// TIA Portal V21 export
FUNCTION_BLOCK "FB303"   // FB303, LAD
TITLE = FB303
{ S7_Optimized_Access := 'TRUE' }
AUTHOR : PRECISE
FAMILY : PRECISE
// SPARGING
// stored: AutoNumber false, MemoryReserve 100, SetENOAutomatically false
   VAR_INPUT
      Enable : Bool;
      Disable : Bool;
      Fault : Bool;
      SecPulse : Bool;
      AlwaysTrue { ExternalVisible := 'False'} : Bool;
      StartConfirmationPopupSel : Bool;   // StartConfirmationPopupSel: 0-NO/1-YES
      EndConfirmationPopupSel : Bool;   // EndConfirmationPopupSel: 0-NO/1-YES
      SpargingModeSel : Int;   // Sparging Mode Selection: 0-DO/1-Time
      SpargingTimebaseSel : Bool;   // Sparging Timebase Selection: 0-sec/1-min
      SpargingLineSel : Bool;   // Sparging LineSelection: 0-THRU GAS FILTER /1-THRU VV
      GasSel : Int;   // Gas Selection - 0-AIR/1-N2
      SetDO : Real := 10.0;   // For Sparging Mode Selection: 0-DO
      SpargingTimeMin : Int := 1;   // For Sparging Mode Selection: 1-Time & Sparging Timebase Selection: 1-min
      SpargingTimeSec : Int := 30;   // For Sparging Mode Selection: 1-Time & Sparging Timebase Selection: 0-sec
      PressuretoOpenVV : Real := 1.0;   // For Sparging LineSelection: 1-THRU VV
      PressuretoCloseVV : Real := 0.5;   // For Sparging LineSelection: 1-THRU VV
      ActualDO : Real;   // For Sparging Mode Selection: 0-DO
      ActualPressure : Real;   // For Sparging LineSelection: 1-THRU VV
      DelaytoOpenGasIn : Int := 3;
   END_VAR
   VAR_OUTPUT
      AirValve : Bool;
      N2Valve : Bool;
      SpargingLineValves : Bool;
      VentValve : Bool;   // For Sparging LineSelection: 1-THRU VV
      StartConfirmationPopup : Bool;   // For Start Confirmation Popup Selection: Yes
      EndConfirmationPopup : Bool;   // For End Confirmation Popup Selection: Yes
      SpargingTimeMinPV : DInt;
      SpargingTimeSecPV : DInt;
      PrintTrigger { ExternalAccessible := 'False'; ExternalVisible := 'False'; ExternalWritable := 'False'} : Bool;
      PrintWord : Int;
      PrintStatus : String[50];
   END_VAR
   VAR_IN_OUT
      Start : Bool;
      Stop : Bool;
      Reset : Bool;
      StartConfirmationAck : Bool;   // For Start Confirmation Popup Selection: Yes
      EndConfirmationAck : Bool;   // For End Confirmation Popup Selection: Yes
      SpareBtn1 : Bool;
      SpareBtn2 : Bool;
      SpareBtn3 : Bool;
      Running : Bool;
      Selected : Bool;
      Paused : Bool;
      StartConfirmationPopupTemp : Bool;   // For Start Confirmation Popup Selection: Yes
      EndConfirmationPopupTemp : Bool;   // For End Confirmation Popup Selection: Yes
      SpargingStarted : Bool;
      SpargingOver : Bool;
      SpargingTimerRunning : Bool;
   END_VAR
   VAR
      ValveOnDelayPV : Int;
      ValveOffDelayPV : Int;
      PrintTriggerTemp : Bool;
      RE1 : Bool;
      RE2 : Bool;
      RE3 : Bool;
      RE4 : Bool;
      RE5 : Bool;
      RE6 : Bool;
      RE7 : Bool;
      SpargingTimer : "FB101";
      PrintTriggerResetTimer { S7_SetPoint := 'True'} : TON_TIME;
      BtnResetTimer { S7_SetPoint := 'True'} : TON_TIME;
   END_VAR
   VAR_TEMP
      STATUS1 : String[40];
      STATUS2 : String[40];
      STATUS3 : String[40];
      STATUS4 : String[40];
      STATUS5 : String[40];
   END_VAR
   VAR_TEMP   // added for the SCL form of the ladder/FBD networks
      _w1 : Bool;
      _w2 : Bool;
      _w3 : Bool;
      _w4 : Bool;
      _w5 : Bool;
   END_VAR
BEGIN

REGION Network 1: Running
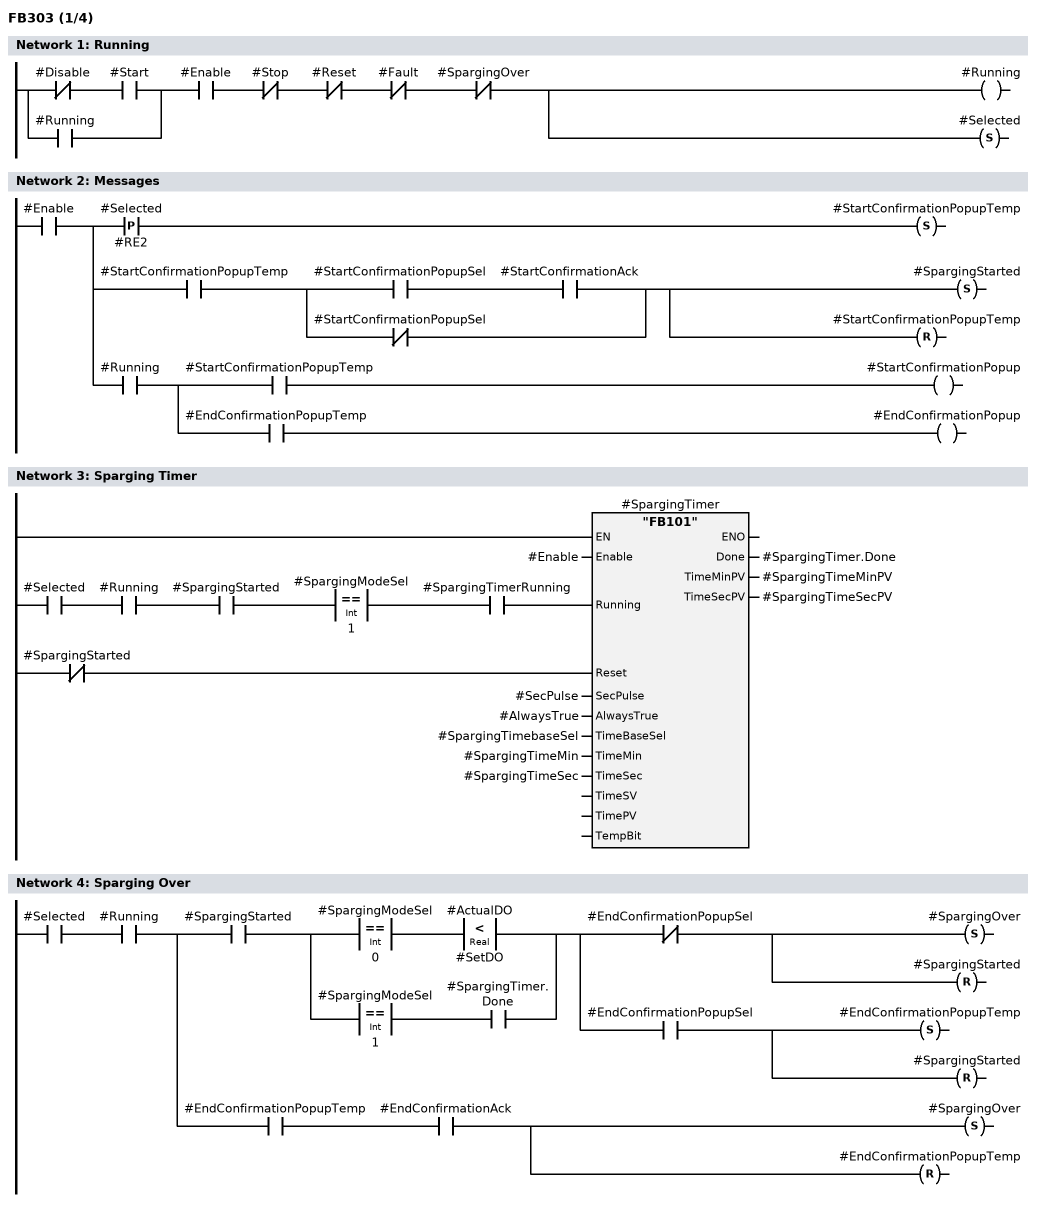
   RUNG wire#powerrail
      I_Contact( #Disable )
      Contact( #Start )
      wire#w1
      Contact( #Enable )
      I_Contact( #Stop )
      I_Contact( #Reset )
      I_Contact( #Fault )
      I_Contact( #SpargingOver )
      wire#w2
      Coil( #Running )
   END_RUNG
   RUNG wire#powerrail
      Contact( #Running )
   END_RUNG wire#w1
   RUNG wire#w2
      S_Coil( #Selected )
   END_RUNG
   // the same network as SCL:
   #Running := ((NOT #Disable AND #Start) OR #Running) AND #Enable AND NOT #Stop AND NOT #Reset AND NOT #Fault AND NOT #SpargingOver;
   IF #Running THEN #Selected := TRUE; END_IF;
END_REGION

REGION Network 2: Messages
   RUNG wire#powerrail
      Contact( #Enable )
      wire#w1
      P_Contact(operand := #Selected, bit := #RE2)
      S_Coil( #StartConfirmationPopupTemp )
   END_RUNG
   RUNG wire#w1
      Contact( #StartConfirmationPopupTemp )
      wire#w2
      Contact( #StartConfirmationPopupSel )
      Contact( #StartConfirmationAck )
      wire#w3
      S_Coil( #SpargingStarted )
   END_RUNG
   RUNG wire#w2
      I_Contact( #StartConfirmationPopupSel )
   END_RUNG wire#w3
   RUNG wire#w3
      R_Coil( #StartConfirmationPopupTemp )
   END_RUNG
   RUNG wire#w1
      Contact( #Running )
      wire#w4
      Contact( #StartConfirmationPopupTemp )
      Coil( #StartConfirmationPopup )
   END_RUNG
   RUNG wire#w4
      Contact( #EndConfirmationPopupTemp )
      Coil( #EndConfirmationPopup )
   END_RUNG
   // the same network as SCL:
   #_w1 := #Enable AND #Selected AND NOT #RE2;   // rising edge of #Selected
   #RE2 := #Selected;
   IF #_w1 THEN #StartConfirmationPopupTemp := TRUE; END_IF;
   IF #Enable AND #StartConfirmationPopupTemp AND ((#StartConfirmationPopupSel AND #StartConfirmationAck) OR NOT #StartConfirmationPopupSel) THEN
       #SpargingStarted := TRUE;
       #StartConfirmationPopupTemp := FALSE;
   END_IF;
   #_w2 := #Enable AND #Running;
   #StartConfirmationPopup := #_w2 AND #StartConfirmationPopupTemp;
   #EndConfirmationPopup := #_w2 AND #EndConfirmationPopupTemp;
END_REGION

REGION Network 3: Sparging Timer
   RUNG wire#powerrail
      #SpargingTimer(Running := wire#w1, Reset := wire#w2, Enable := #Enable, SecPulse := #SecPulse, AlwaysTrue := #AlwaysTrue, TimeBaseSel := #SpargingTimebaseSel, TimeMin := #SpargingTimeMin, TimeSec := #SpargingTimeSec, TimeSV :=, TimePV :=, TempBit :=, Done => #SpargingTimer.Done, TimeMinPV => #SpargingTimeMinPV, TimeSecPV => #SpargingTimeSecPV)
   END_RUNG
   RUNG wire#powerrail
      Contact( #Selected )
      Contact( #Running )
      Contact( #SpargingStarted )
      { S7_Templates := "SrcType := Int" } EQ_Contact(in1 := #SpargingModeSel, in2 := 1)
      Contact( #SpargingTimerRunning )
   END_RUNG wire#w1
   RUNG wire#powerrail
      I_Contact( #SpargingStarted )
   END_RUNG wire#w2
   // the same network as SCL:
   #SpargingTimer(Enable := #Enable,   // "FB101"
                  Running := #Selected AND #Running AND #SpargingStarted AND (#SpargingModeSel = 1) AND #SpargingTimerRunning,
                  Reset := NOT #SpargingStarted,
                  SecPulse := #SecPulse,
                  AlwaysTrue := #AlwaysTrue,
                  TimeBaseSel := #SpargingTimebaseSel,
                  TimeMin := #SpargingTimeMin,
                  TimeSec := #SpargingTimeSec,
                  Done => #SpargingTimer.Done,
                  TimeMinPV => #SpargingTimeMinPV,
                  TimeSecPV => #SpargingTimeSecPV);
END_REGION

REGION Network 4: Sparging Over
   RUNG wire#powerrail
      Contact( #Selected )
      Contact( #Running )
      wire#w1
      Contact( #SpargingStarted )
      wire#w2
      { S7_Templates := "SrcType := Int" } EQ_Contact(in1 := #SpargingModeSel, in2 := 0)
      { S7_Templates := "SrcType := Real" } LT_Contact(in1 := #ActualDO, in2 := #SetDO)
      wire#w3
      I_Contact( #EndConfirmationPopupSel )
      wire#w4
      S_Coil( #SpargingOver )
   END_RUNG
   RUNG wire#w2
      { S7_Templates := "SrcType := Int" } EQ_Contact(in1 := #SpargingModeSel, in2 := 1)
      Contact( #SpargingTimer.Done )
   END_RUNG wire#w3
   RUNG wire#w4
      R_Coil( #SpargingStarted )
   END_RUNG
   RUNG wire#w3
      Contact( #EndConfirmationPopupSel )
      wire#w5
      S_Coil( #EndConfirmationPopupTemp )
   END_RUNG
   RUNG wire#w5
      R_Coil( #SpargingStarted )
   END_RUNG
   RUNG wire#w1
      Contact( #EndConfirmationPopupTemp )
      Contact( #EndConfirmationAck )
      wire#w6
      S_Coil( #SpargingOver )
   END_RUNG
   RUNG wire#w6
      R_Coil( #EndConfirmationPopupTemp )
   END_RUNG
   // the same network as SCL:
   #_w1 := #Selected AND #Running;
   #_w2 := #_w1 AND #SpargingStarted AND (((#SpargingModeSel = 0) AND (#ActualDO < #SetDO)) OR ((#SpargingModeSel = 1) AND #SpargingTimer.Done));
   IF #_w2 AND NOT #EndConfirmationPopupSel THEN
       #SpargingOver := TRUE;
       #SpargingStarted := FALSE;
   END_IF;
   IF #_w2 AND #EndConfirmationPopupSel THEN
       #EndConfirmationPopupTemp := TRUE;
       #SpargingStarted := FALSE;
   END_IF;
   IF #_w1 AND #EndConfirmationPopupTemp AND #EndConfirmationAck THEN
       #SpargingOver := TRUE;
       #EndConfirmationPopupTemp := FALSE;
   END_IF;
END_REGION

REGION Network 5: Output On
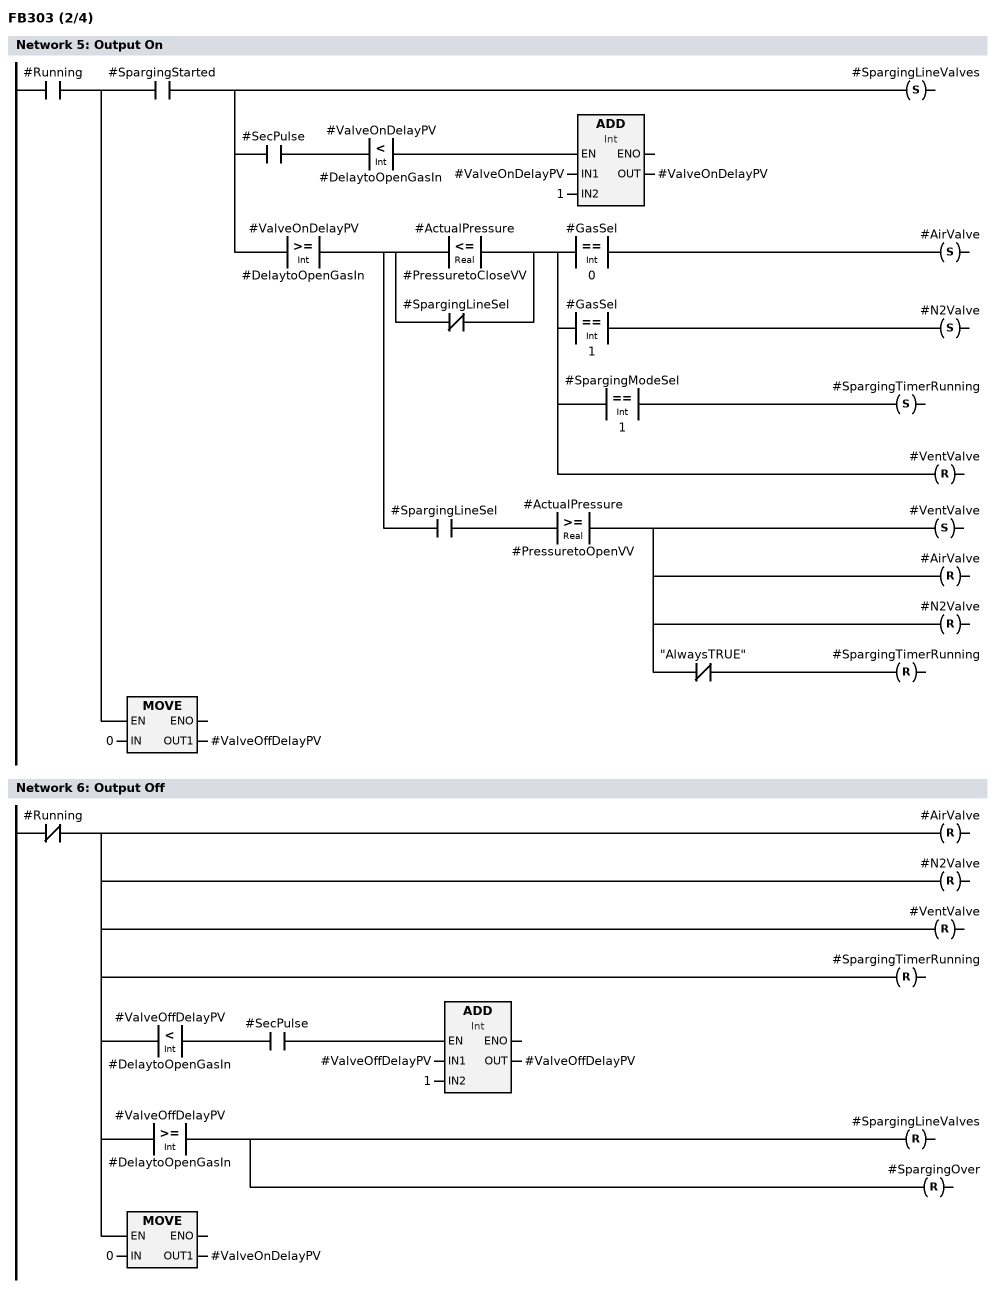
   RUNG wire#powerrail
      Contact( #Running )
      wire#w1
      Contact( #SpargingStarted )
      wire#w2
      S_Coil( #SpargingLineValves )
   END_RUNG
   RUNG wire#w2
      Contact( #SecPulse )
      { S7_Templates := "SrcType := Int" } LT_Contact(in1 := #ValveOnDelayPV, in2 := #DelaytoOpenGasIn)
      { S7_Templates := "SrcType := Int"; S7_GenerateENO := "TRUE" } Add(in1 := #ValveOnDelayPV, in2 := 1, out => #ValveOnDelayPV)
   END_RUNG
   RUNG wire#w2
      { S7_Templates := "SrcType := Int" } GE_Contact(in1 := #ValveOnDelayPV, in2 := #DelaytoOpenGasIn)
      wire#w3
      { S7_Templates := "SrcType := Real" } LE_Contact(in1 := #ActualPressure, in2 := #PressuretoCloseVV)
      wire#w4
      { S7_Templates := "SrcType := Int" } EQ_Contact(in1 := #GasSel, in2 := 0)
      S_Coil( #AirValve )
   END_RUNG
   RUNG wire#w3
      I_Contact( #SpargingLineSel )
   END_RUNG wire#w4
   RUNG wire#w4
      { S7_Templates := "SrcType := Int" } EQ_Contact(in1 := #GasSel, in2 := 1)
      S_Coil( #N2Valve )
   END_RUNG
   RUNG wire#w4
      { S7_Templates := "SrcType := Int" } EQ_Contact(in1 := #SpargingModeSel, in2 := 1)
      S_Coil( #SpargingTimerRunning )
   END_RUNG
   RUNG wire#w4
      R_Coil( #VentValve )
   END_RUNG
   RUNG wire#w3
      Contact( #SpargingLineSel )
      { S7_Templates := "SrcType := Real" } GE_Contact(in1 := #ActualPressure, in2 := #PressuretoOpenVV)
      wire#w5
      S_Coil( #VentValve )
   END_RUNG
   RUNG wire#w5
      R_Coil( #AirValve )
   END_RUNG
   RUNG wire#w5
      R_Coil( #N2Valve )
   END_RUNG
   RUNG wire#w5
      I_Contact( "AlwaysTRUE" )
      R_Coil( #SpargingTimerRunning )
   END_RUNG
   RUNG wire#w1
      { S7_GenerateENO := "TRUE" } Move(in := 0, out1 => #ValveOffDelayPV)
   END_RUNG
   // the same network as SCL:
   #_w1 := #Running AND #SpargingStarted;
   IF #_w1 THEN #SpargingLineValves := TRUE; END_IF;
   IF #_w1 AND #SecPulse AND (#ValveOnDelayPV < #DelaytoOpenGasIn) THEN
       #ValveOnDelayPV := #ValveOnDelayPV + 1;
   END_IF;
   #_w2 := #_w1 AND (#ValveOnDelayPV >= #DelaytoOpenGasIn);
   #_w3 := #_w2 AND ((#ActualPressure <= #PressuretoCloseVV) OR NOT #SpargingLineSel);
   IF #_w3 AND (#GasSel = 0) THEN #AirValve := TRUE; END_IF;
   IF #_w3 AND (#GasSel = 1) THEN #N2Valve := TRUE; END_IF;
   IF #_w3 AND (#SpargingModeSel = 1) THEN #SpargingTimerRunning := TRUE; END_IF;
   IF #_w3 THEN #VentValve := FALSE; END_IF;
   #_w4 := #_w2 AND #SpargingLineSel AND (#ActualPressure >= #PressuretoOpenVV);
   IF #_w4 THEN
       #VentValve := TRUE;
       #AirValve := FALSE;
       #N2Valve := FALSE;
   END_IF;
   IF #_w4 AND NOT "AlwaysTRUE" THEN #SpargingTimerRunning := FALSE; END_IF;
   IF #Running THEN #ValveOffDelayPV := 0; END_IF;
END_REGION

REGION Network 6: Output Off
   RUNG wire#powerrail
      I_Contact( #Running )
      wire#w1
      R_Coil( #AirValve )
   END_RUNG
   RUNG wire#w1
      R_Coil( #N2Valve )
   END_RUNG
   RUNG wire#w1
      R_Coil( #VentValve )
   END_RUNG
   RUNG wire#w1
      R_Coil( #SpargingTimerRunning )
   END_RUNG
   RUNG wire#w1
      { S7_Templates := "SrcType := Int" } LT_Contact(in1 := #ValveOffDelayPV, in2 := #DelaytoOpenGasIn)
      Contact( #SecPulse )
      { S7_Templates := "SrcType := Int"; S7_GenerateENO := "TRUE" } Add(in1 := #ValveOffDelayPV, in2 := 1, out => #ValveOffDelayPV)
   END_RUNG
   RUNG wire#w1
      { S7_Templates := "SrcType := Int" } GE_Contact(in1 := #ValveOffDelayPV, in2 := #DelaytoOpenGasIn)
      wire#w2
      R_Coil( #SpargingLineValves )
   END_RUNG
   RUNG wire#w2
      R_Coil( #SpargingOver )
   END_RUNG
   RUNG wire#w1
      { S7_GenerateENO := "TRUE" } Move(in := 0, out1 => #ValveOnDelayPV)
   END_RUNG
   // the same network as SCL:
   IF NOT #Running THEN
       #AirValve := FALSE;
       #N2Valve := FALSE;
       #VentValve := FALSE;
       #SpargingTimerRunning := FALSE;
   END_IF;
   IF NOT #Running AND (#ValveOffDelayPV < #DelaytoOpenGasIn) AND #SecPulse THEN
       #ValveOffDelayPV := #ValveOffDelayPV + 1;
   END_IF;
   IF NOT #Running AND (#ValveOffDelayPV >= #DelaytoOpenGasIn) THEN
       #SpargingLineValves := FALSE;
       #SpargingOver := FALSE;
   END_IF;
   IF NOT #Running THEN #ValveOnDelayPV := 0; END_IF;
END_REGION

REGION Network 7: Event Status
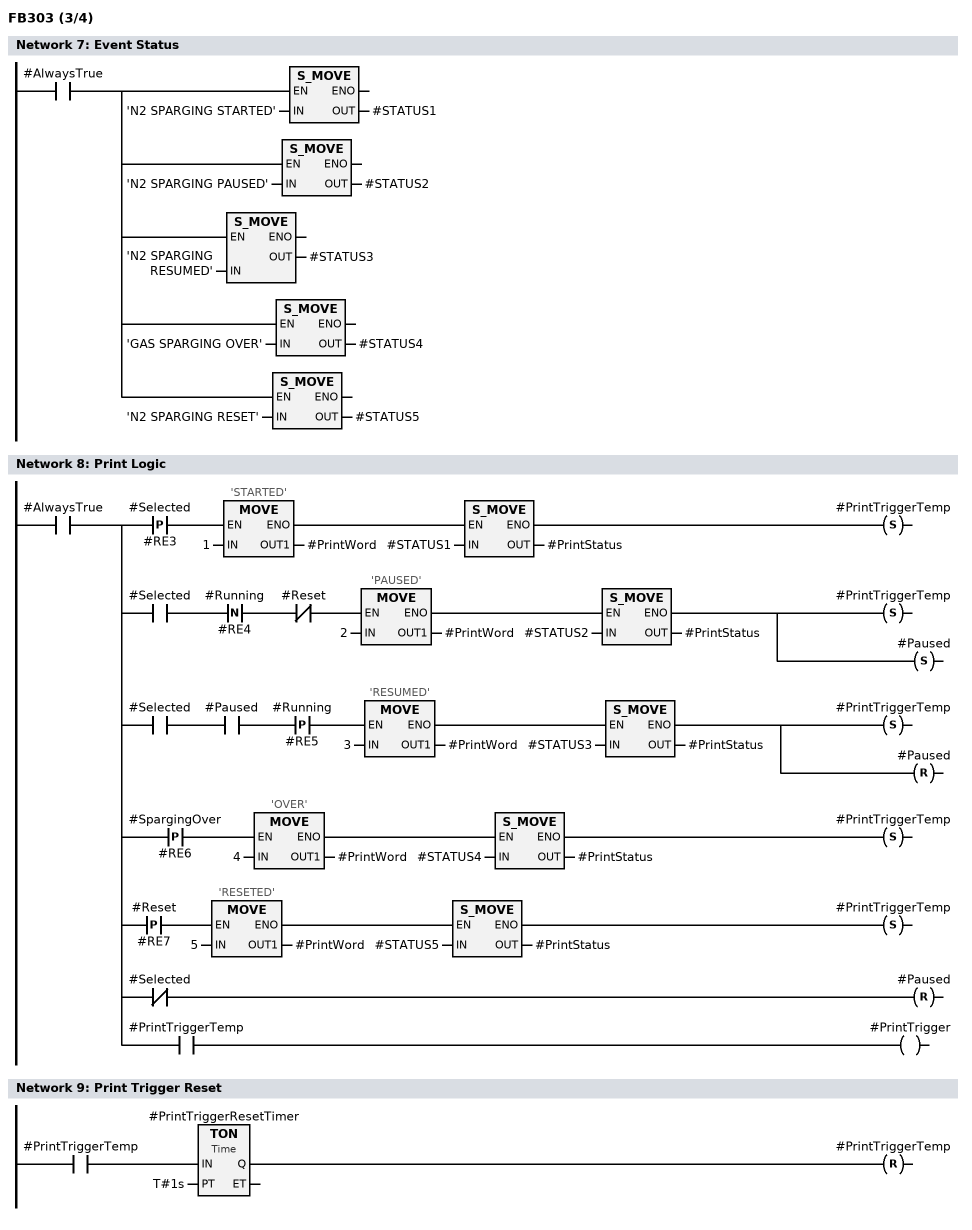
   RUNG wire#powerrail
      Contact( #AlwaysTrue )
      wire#w1
      S_Move(in := 'N2 SPARGING STARTED', out => #STATUS1)
   END_RUNG
   RUNG wire#w1
      S_Move(in := 'N2 SPARGING PAUSED', out => #STATUS2)
   END_RUNG
   RUNG wire#w1
      S_Move(in := 'N2 SPARGING RESUMED', out => #STATUS3)
   END_RUNG
   RUNG wire#w1
      S_Move(in := 'GAS SPARGING OVER', out => #STATUS4)
   END_RUNG
   RUNG wire#w1
      S_Move(in := 'N2 SPARGING RESET', out => #STATUS5)
   END_RUNG
   // the same network as SCL:
   IF #AlwaysTrue THEN
       #STATUS1 := 'N2 SPARGING STARTED';
       #STATUS2 := 'N2 SPARGING PAUSED';
       #STATUS3 := 'N2 SPARGING RESUMED';
       #STATUS4 := 'GAS SPARGING OVER';
       #STATUS5 := 'N2 SPARGING RESET';
   END_IF;
END_REGION

REGION Network 8: Print Logic
   RUNG wire#powerrail
      Contact( #AlwaysTrue )
      wire#w1
      P_Contact(operand := #Selected, bit := #RE3)
      { S7_GenerateENO := "TRUE" } Move(in := 1, out1 => #PrintWord)   // 'STARTED'
      S_Move(in := #STATUS1, out => #PrintStatus)
      S_Coil( #PrintTriggerTemp )
   END_RUNG
   RUNG wire#w1
      Contact( #Selected )
      N_Contact(operand := #Running, bit := #RE4)
      I_Contact( #Reset )
      { S7_GenerateENO := "TRUE" } Move(in := 2, out1 => #PrintWord)   // 'PAUSED'
      S_Move(in := #STATUS2, out => #PrintStatus)
      wire#w2
      S_Coil( #PrintTriggerTemp )
   END_RUNG
   RUNG wire#w2
      S_Coil( #Paused )
   END_RUNG
   RUNG wire#w1
      Contact( #Selected )
      Contact( #Paused )
      P_Contact(operand := #Running, bit := #RE5)
      { S7_GenerateENO := "TRUE" } Move(in := 3, out1 => #PrintWord)   // 'RESUMED'
      S_Move(in := #STATUS3, out => #PrintStatus)
      wire#w3
      S_Coil( #PrintTriggerTemp )
   END_RUNG
   RUNG wire#w3
      R_Coil( #Paused )
   END_RUNG
   RUNG wire#w1
      P_Contact(operand := #SpargingOver, bit := #RE6)
      { S7_GenerateENO := "TRUE" } Move(in := 4, out1 => #PrintWord)   // 'OVER'
      S_Move(in := #STATUS4, out => #PrintStatus)
      S_Coil( #PrintTriggerTemp )
   END_RUNG
   RUNG wire#w1
      P_Contact(operand := #Reset, bit := #RE7)
      { S7_GenerateENO := "TRUE" } Move(in := 5, out1 => #PrintWord)   // 'RESETED'
      S_Move(in := #STATUS5, out => #PrintStatus)
      S_Coil( #PrintTriggerTemp )
   END_RUNG
   RUNG wire#w1
      I_Contact( #Selected )
      R_Coil( #Paused )
   END_RUNG
   RUNG wire#w1
      Contact( #PrintTriggerTemp )
      Coil( #PrintTrigger )
   END_RUNG
   // the same network as SCL:
   // ENO of a box is taken as its EN; it also drops when the box reports an error
   #_w1 := #AlwaysTrue AND #Selected AND NOT #RE3;   // rising edge of #Selected
   #RE3 := #Selected;
   IF #_w1 THEN
       #PrintWord := 1;   // 'STARTED'
       #PrintStatus := #STATUS1;
       #PrintTriggerTemp := TRUE;
   END_IF;
   #_w2 := #AlwaysTrue AND #Selected AND NOT #Running AND #RE4;   // falling edge of #Running
   #RE4 := #Running;
   IF #_w2 AND NOT #Reset THEN
       #PrintWord := 2;   // 'PAUSED'
       #PrintStatus := #STATUS2;
       #PrintTriggerTemp := TRUE;
       #Paused := TRUE;
   END_IF;
   #_w3 := #AlwaysTrue AND #Selected AND #Paused AND #Running AND NOT #RE5;   // rising edge of #Running
   #RE5 := #Running;
   IF #_w3 THEN
       #PrintWord := 3;   // 'RESUMED'
       #PrintStatus := #STATUS3;
       #PrintTriggerTemp := TRUE;
       #Paused := FALSE;
   END_IF;
   #_w4 := #AlwaysTrue AND #SpargingOver AND NOT #RE6;   // rising edge of #SpargingOver
   #RE6 := #SpargingOver;
   IF #_w4 THEN
       #PrintWord := 4;   // 'OVER'
       #PrintStatus := #STATUS4;
       #PrintTriggerTemp := TRUE;
   END_IF;
   #_w5 := #AlwaysTrue AND #Reset AND NOT #RE7;   // rising edge of #Reset
   #RE7 := #Reset;
   IF #_w5 THEN
       #PrintWord := 5;   // 'RESETED'
       #PrintStatus := #STATUS5;
       #PrintTriggerTemp := TRUE;
   END_IF;
   IF #AlwaysTrue AND NOT #Selected THEN #Paused := FALSE; END_IF;
   #PrintTrigger := #AlwaysTrue AND #PrintTriggerTemp;
END_REGION

REGION Network 9: Print Trigger Reset
   RUNG wire#powerrail
      Contact( #PrintTriggerTemp )
      { S7_Templates := "time_type := Time" } #PrintTriggerResetTimer.TON(pt := T#1s, et =>)
      R_Coil( #PrintTriggerTemp )
   END_RUNG
   // the same network as SCL:
   #PrintTriggerResetTimer(IN := #PrintTriggerTemp, PT := T#1s);   // TON
   IF #PrintTriggerResetTimer.Q THEN #PrintTriggerTemp := FALSE; END_IF;
END_REGION

REGION Network 10: Button Reset
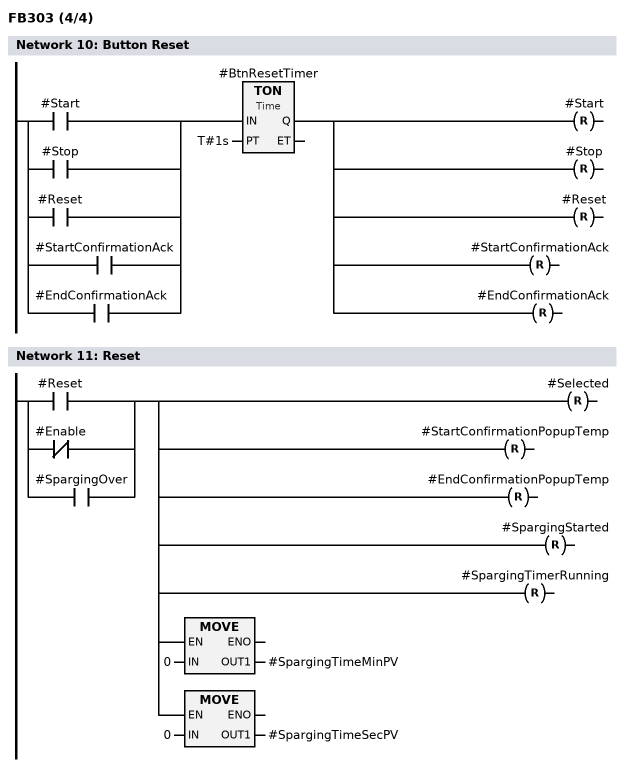
   RUNG wire#powerrail
      Contact( #Start )
      wire#w1
      { S7_Templates := "time_type := Time" } #BtnResetTimer.TON(pt := T#1s, et =>)
      wire#w2
      R_Coil( #Start )
   END_RUNG
   RUNG wire#powerrail
      Contact( #Stop )
   END_RUNG wire#w1
   RUNG wire#powerrail
      Contact( #Reset )
   END_RUNG wire#w1
   RUNG wire#powerrail
      Contact( #StartConfirmationAck )
   END_RUNG wire#w1
   RUNG wire#powerrail
      Contact( #EndConfirmationAck )
   END_RUNG wire#w1
   RUNG wire#w2
      R_Coil( #Stop )
   END_RUNG
   RUNG wire#w2
      R_Coil( #Reset )
   END_RUNG
   RUNG wire#w2
      R_Coil( #StartConfirmationAck )
   END_RUNG
   RUNG wire#w2
      R_Coil( #EndConfirmationAck )
   END_RUNG
   // the same network as SCL:
   #BtnResetTimer(IN := #Start OR #Stop OR #Reset OR #StartConfirmationAck OR #EndConfirmationAck, PT := T#1s);   // TON
   IF #BtnResetTimer.Q THEN
       #Start := FALSE;
       #Stop := FALSE;
       #Reset := FALSE;
       #StartConfirmationAck := FALSE;
       #EndConfirmationAck := FALSE;
   END_IF;
END_REGION

REGION Network 11: Reset
   RUNG wire#powerrail
      Contact( #Reset )
      wire#w1
      R_Coil( #Selected )
   END_RUNG
   RUNG wire#powerrail
      I_Contact( #Enable )
   END_RUNG wire#w1
   RUNG wire#powerrail
      Contact( #SpargingOver )
   END_RUNG wire#w1
   RUNG wire#w1
      R_Coil( #StartConfirmationPopupTemp )
   END_RUNG
   RUNG wire#w1
      R_Coil( #EndConfirmationPopupTemp )
   END_RUNG
   RUNG wire#w1
      R_Coil( #SpargingStarted )
   END_RUNG
   RUNG wire#w1
      R_Coil( #SpargingTimerRunning )
   END_RUNG
   RUNG wire#w1
      { S7_GenerateENO := "TRUE" } Move(in := 0, out1 => #SpargingTimeMinPV)
   END_RUNG
   RUNG wire#w1
      { S7_GenerateENO := "TRUE" } Move(in := 0, out1 => #SpargingTimeSecPV)
   END_RUNG
   // the same network as SCL:
   IF #Reset OR NOT #Enable OR #SpargingOver THEN
       #Selected := FALSE;
       #StartConfirmationPopupTemp := FALSE;
       #EndConfirmationPopupTemp := FALSE;
       #SpargingStarted := FALSE;
       #SpargingTimerRunning := FALSE;
       #SpargingTimeMinPV := 0;
       #SpargingTimeSecPV := 0;
   END_IF;
END_REGION
END_FUNCTION_BLOCK
